(* IEC 61131-3 sources: repolevel_ST_code_completion/dataset/generation_context_ground_truth/plc_hello_mixing_tank, 4 files *)

(* ---- F_ResetDeviceCommands.st ---- *)
// 命令合理性复位
// 当设备到达目标状态时，复位相应的命令标志

// 混合电机命令复位
IF bMixerRunning THEN
	bMixerRunCmd := FALSE;		// 已运行，复位运行命令
ELSE
	bMixerStopCmd := FALSE;		// 已停止，复位停止命令
END_IF

// 介质1阀门命令复位
IF bMedium1Opened THEN
	bMedium1OpenCmd := FALSE;	// 已打开，复位打开命令
ELSE
	bMedium1CloseCmd := FALSE;	// 已关闭，复位关闭命令
END_IF

// 介质2阀门命令复位
IF bMedium2Opened THEN
	bMedium2OpenCmd := FALSE;	// 已打开，复位打开命令
ELSE
	bMedium2CloseCmd := FALSE;	// 已关闭，复位关闭命令
END_IF

// 排空阀门命令复位
IF bDrainOpened THEN
	bDrainOpenCmd := FALSE;		// 已打开，复位打开命令
ELSE
	bDrainCloseCmd := FALSE;	// 已关闭，复位关闭命令
END_IF

F_ResetDeviceCommands := TRUE;

(* ---- FB_AutoSequence.st ---- *)
VAR
	tonMixing			:	TON;			// 混合定时器
END_VAR

// 复位逻辑
IF bReset THEN
	eCurrentState := AUTO_SEQUENCE.DRAINING;
	nCyclesCompleted := 0;
END_IF

// 自动序列状态机
IF bEnable THEN
	CASE eCurrentState OF
		AUTO_SEQUENCE.FILLING:
			// 确保其他设备不工作
			bMixerRunCmd := FALSE;
			bDrainOpenCmd := FALSE;

			// 打开两个介质阀门，开始填充罐体
			bMedium1OpenCmd := NOT bTankLevelFull;
			bMedium2OpenCmd := NOT bTankLevelFull;

			// 当罐体满时，等待填充阀关闭，然后进入混合状态
			IF bTankLevelFull AND NOT (bMedium1Opened OR bMedium2Opened) THEN
				eCurrentState := AUTO_SEQUENCE.MIXING;
			END_IF

		AUTO_SEQUENCE.MIXING:
			// 确保其他设备不工作
			bMedium1OpenCmd := FALSE;
			bMedium2OpenCmd := FALSE;
			bDrainOpenCmd := FALSE;

			// 启动混合电机并混合10秒
			bMixerRunCmd := TRUE;
			tonMixing(IN := bMixerRunning, PT := tMixingDuration);

			// 当定时器到达10秒，等待电机停止运行，然后进入排空状态
			IF tonMixing.Q THEN
				bMixerRunCmd := FALSE;
				eCurrentState := AUTO_SEQUENCE.DRAINING;
			END_IF

		AUTO_SEQUENCE.DRAINING:
			// 确保其他设备不工作
			bMixerRunCmd := FALSE;
			bMedium1OpenCmd := FALSE;
			bMedium2OpenCmd := FALSE;

			// 打开排空阀，开始排空罐体
			bDrainOpenCmd := NOT bTankLevelEmpty;

			// 当罐体空时，等待排空阀关闭，然后进入填充状态
			IF bTankLevelEmpty AND NOT bDrainOpened THEN
				eCurrentState := AUTO_SEQUENCE.FILLING;
				nCyclesCompleted := nCyclesCompleted + 1;
			END_IF
	END_CASE
ELSE
	// 禁用时，关闭所有输出
	bMixerRunCmd := FALSE;
	bMedium1OpenCmd := FALSE;
	bMedium2OpenCmd := FALSE;
	bDrainOpenCmd := FALSE;
	tonMixing(IN := FALSE);
END_IF

(* ---- FB_ModeController.st ---- *)
VAR
	eLastMode		:	MODES;	// 上次模式
END_VAR

// 模式切换逻辑
CASE eCurrentMode OF
	MODES.AUTO:
		IF bSetToManual THEN
			eCurrentMode := MODES.MANUAL;
		END_IF

	MODES.MANUAL:
		IF bSetToAuto THEN
			eCurrentMode := MODES.AUTO;
		END_IF
END_CASE

// 检测模式变化
bModeChanged := (eCurrentMode <> eLastMode);
eLastMode := eCurrentMode;

(* ---- FB_TankLevelSimulator.st ---- *)
// 复位逻辑
IF bReset THEN
	rCurrentLevel := rInitialLevel;
END_IF

// 液位计算
// 如果任一填充阀打开则填充，如果排空阀打开则排空
rCurrentLevel := rCurrentLevel
				+ rFillRate1 * BOOL_TO_REAL(bMedium1Opened)
				+ rFillRate2 * BOOL_TO_REAL(bMedium2Opened)
				- rDrainRate * BOOL_TO_REAL(bDrainOpened);

// 限制液位范围 (0-100%)
rCurrentLevel := LIMIT(rMinLevel, rCurrentLevel, rMaxLevel);
